// Examples of collectors.
// [Hint]
// > All reference-variables are implemented to ease monitoring of relevant variables.
FUNCTION_BLOCK FB_Ref_Collectors EXTENDS FB_BA_View
VAR
	{region 'Analog'}
		_ValueA1					: REFERENCE TO REAL				REF= ValueA1.fValueRm;
		ValueA1						: FB_BA_AV_Op := (
										iParent						:= THIS^,
										iProfile					:= MyProfiles.AVOp_Prf,
										fValueRm					:= 0.0
									);
		_ValueA2					: REFERENCE TO REAL				REF= ValueA2.fValueRm;
		ValueA2						: FB_BA_AV_Op := (
										iParent						:= THIS^,
										iProfile					:= MyProfiles.AVOp_Prf,
										fValueRm					:= 1.0
									);
		ColectA						: FB_BA_Collector				:= (iParent:=THIS^, iReferences:=[ ValueA1, ValueA2 ]);
	{endregion}
	{region 'Binary'}
		_ValueB1					: REFERENCE TO BOOL				REF= ValueB1.bValueRm;
		ValueB1						: FB_BA_BV_Op := (
										iParent						:= THIS^,
										iProfile					:= MyProfiles.BVOp_Prf,
										bValueRm					:= FALSE
									);
		_ValueB2					: REFERENCE TO BOOL				REF= ValueB2.bValueRm;
		ValueB2						: FB_BA_BV_Op := (
										iParent						:= THIS^,
										iProfile					:= MyProfiles.BVOp_Prf,
										bValueRm					:= TRUE
									);
		ColectB						: FB_BA_Collector				:= (iParent:=THIS^, iReferences:=[ ValueB1, ValueB2 ]);
	{endregion}
	{region 'Multistate'}
		_ValueM1					: REFERENCE TO UDINT			REF= ValueM1.nValueRm;
		ValueM1						: FB_BA_MV_Op := (
										iParent						:= THIS^,
										iProfile					:= MyProfiles.MVOp_Prf,
										nValueRm					:= 1
									);
		_ValueM2					: REFERENCE TO UDINT			REF= ValueM2.nValueRm;
		ValueM2						: FB_BA_MV_Op := (
										iParent						:= THIS^,
										iProfile					:= MyProfiles.MVOp_Prf,
										nValueRm					:= 2
									);
		ColectM						: FB_BA_Collector				:= (iParent:=THIS^, iReferences:=[ ValueM1, ValueM2 ]);
	{endregion}
	{region 'View'}
		View1						: FB_BA_View					:= (iParent:=THIS^, sObjectName:='View1');
			_Enable1				: REFERENCE TO BOOL				REF= Enable1.bValueRm;	
			Enable1					: FB_BA_BV_Op := (
										iParent						:= View1,
										iProfile					:= MyProfiles.BVOp_Prf,
										bValueRm					:= FALSE
									);
			_Value1					: REFERENCE TO REAL				REF= Value1.fValueRm;
			Value1					: FB_BA_AV_Op := (
										iParent						:= View1,
										iProfile					:= MyProfiles.AVOp_Prf,
										fValueRm					:= 0.0
									);
		View2						: FB_BA_View					:= (iParent:=THIS^, sObjectName:='View2');
			_Enable01				: REFERENCE TO BOOL				REF= Enable01.bValueRm;	
			Enable01				: FB_BA_BV_Op := (
										iParent						:= View2,
										iProfile					:= MyProfiles.BVOp_Prf,
										bValueRm					:= TRUE
									);
			_Value01				: REFERENCE TO REAL				REF= Value01.fValueRm;
			Value01					: FB_BA_AV_Op := (
										iParent						:= View2,
										iProfile					:= MyProfiles.AVOp_Prf,
										fValueRm					:= 3.0
									);
		View3						: FB_NestedView					:= (View:=(iParent:=THIS^, sObjectName:='View3'));
			_Enable3				: REFERENCE TO BOOL				REF= View3.Enable.bValueRm;
			_Value3					: REFERENCE TO REAL				REF= View3.Value.fValueRm;
		View4						: FB_SubNestedView				:= (iParent:=THIS^, sObjectName:='View4');
			_Enable4				: REFERENCE TO BOOL				REF= View4.SubView.Enable.bValueRm;
			_Value4					: REFERENCE TO REAL				REF= View4.SubView.Value.fValueRm;
					  
		ColectEnA					: FB_BA_Collector := (
										iParent						:= THIS^,
										iReferences					:= [ View1, View2, View3.View ],
					  					sRefSubjectEn				:= 'Enable',							// <- Specified subject.
					  					sRefSubjectVal				:= 'Value'								// <- Specified subject.
									);
		ColectEnB					: FB_BA_Collector := (
										iParent						:= THIS^,
										iReferences					:= [ View4 ],
					  					sRefSubjectEn				:= 'SubView.Enable',					// <- Specified subject path.
					  					sRefSubjectVal				:= 'SubView.Value'						// <- Specified subject path.
									);
	{endregion}
END_VAR

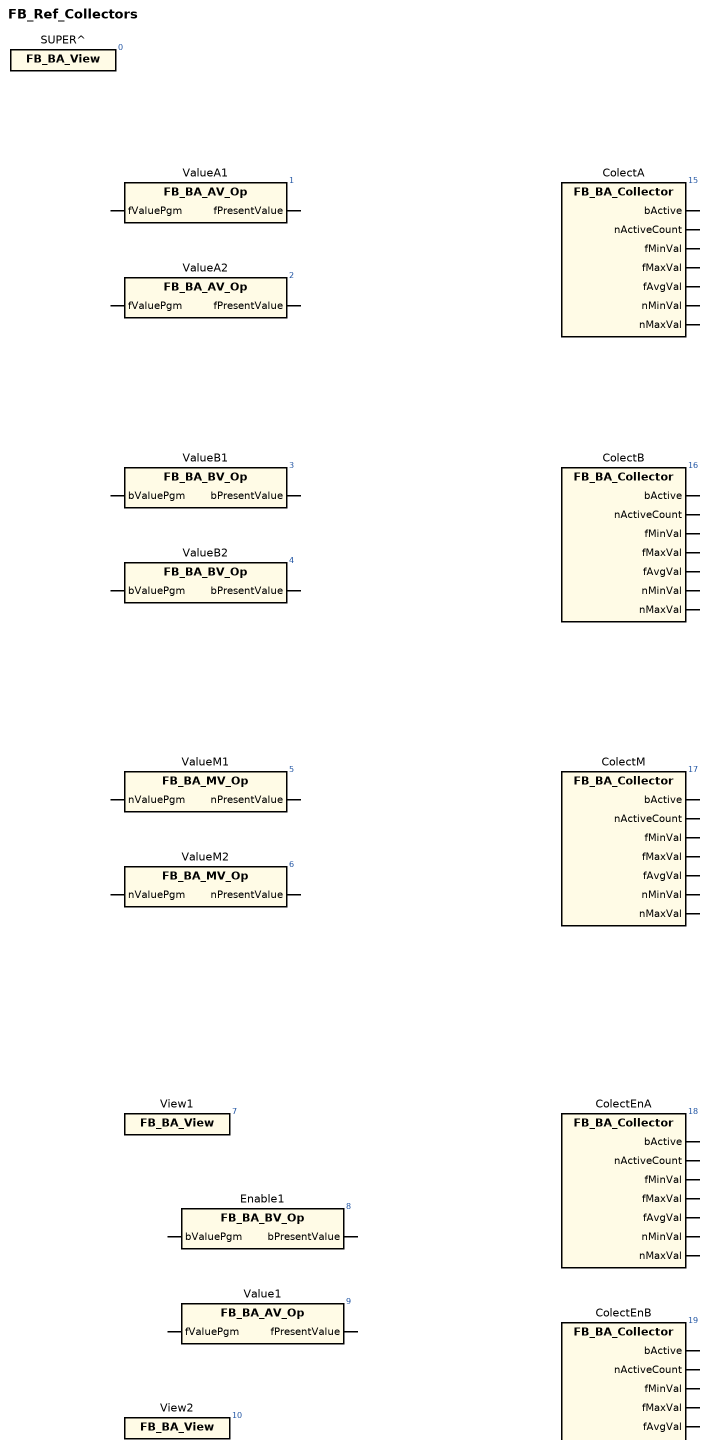
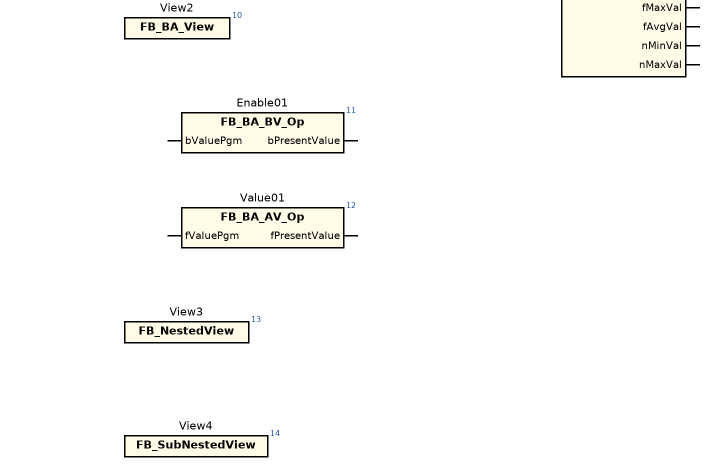
SUPER^(); // FB_BA_View
ValueA1(); // FB_BA_AV_Op
ValueA2(); // FB_BA_AV_Op
ValueB1(); // FB_BA_BV_Op
ValueB2(); // FB_BA_BV_Op
ValueM1(); // FB_BA_MV_Op
ValueM2(); // FB_BA_MV_Op
View1(); // FB_BA_View
Enable1(); // FB_BA_BV_Op
Value1(); // FB_BA_AV_Op
View2(); // FB_BA_View
Enable01(); // FB_BA_BV_Op
Value01(); // FB_BA_AV_Op
View3(); // FB_NestedView
View4(); // FB_SubNestedView
ColectA(); // FB_BA_Collector
ColectB(); // FB_BA_Collector
ColectM(); // FB_BA_Collector
ColectEnA(); // FB_BA_Collector
ColectEnB(); // FB_BA_Collector

END_FUNCTION_BLOCK

(* stored: Version 1.1.0.1, ProductVersion 3.1.4024.5
   POU FB_Ref_Collectors: Id {a36f31c6-10f0-40fb-88e5-72c64b84c691}, SpecialFunc None *)
